PROGRAM MAIN
VAR
	bOut1 : BOOL;
	bOut2 : BOOL;
	iNumber : INT := 50;
	stStruct : stStruct;
END_VAR

bOut1 := Globals.bBool1;
bOut2 := Globals.bBool2;
stStruct.bFirst := TRUE;
stStruct.iSecond := 5;
stStruct.rThird := 1.3;

END_PROGRAM

(* stored: Version 1.1.0.1, ProductVersion 3.1.4024.12
   POU MAIN: Id {cf941a6b-9326-430a-881a-5e529de028d0}, SpecialFunc None *)
